RoboDK station: bokssim.rdk

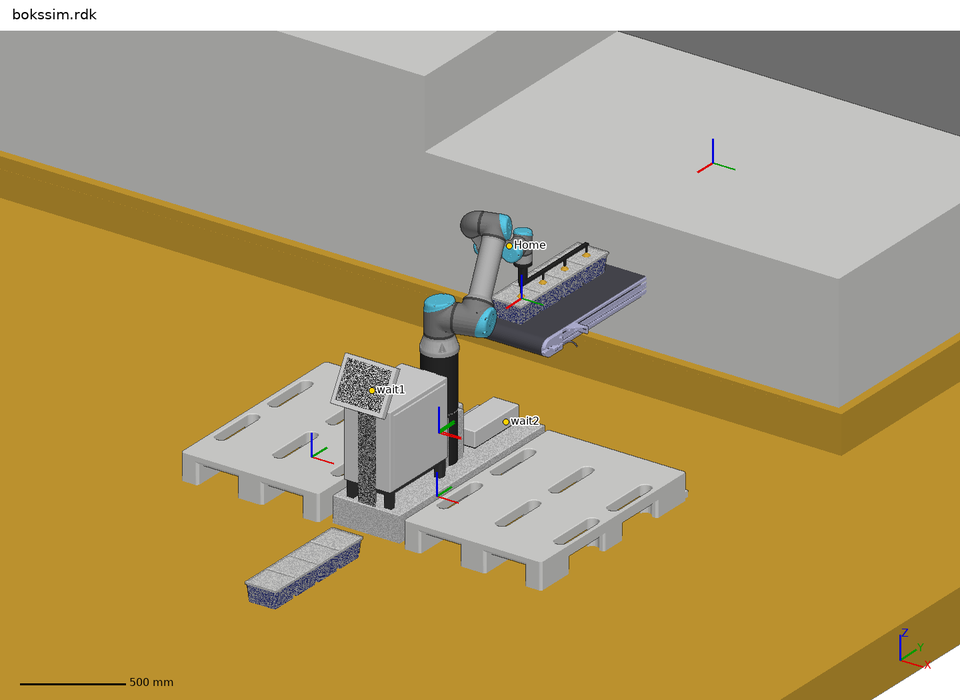
[picture v0: the station drawn from its stored meshes, robots at their saved joint values, targets as dots, program paths as lines]
Station robotsim1. Poses are relative to the parent item; angles as X-Y-Z fixed-axis rotations.
  - object pallPlast-v2 at (-1010, 360, 0) mm, size 800 x 1200 x 150 mm, geometry from pallPlast-v2.step
  - frame Conveyor Belt Base at (-200, 3610, 605) mm, rotated rx 0 ry 0 rz -90 deg
    - robot Conveyor Belt: 1 axes
        modified DH rows (alpha deg, a mm, theta deg, d mm): 0, 0, 0, 0 linear
        base shift (0, 0, 0) mm, rotated rx 0 ry 90 rz 0 deg
        joint limits [-500000] to [500000]; home [0]; saved at [0]
  - object pallPlast-v2 at (280, 360, 0) mm, size 800 x 1200 x 150 mm, geometry from pallPlast-v2.step
  - frame UR16e Base at (40, 1000, 300) mm
    - frame placeFrame at (-380, -510, -40) mm
    - frame placeFrame2 at (350, -520, -40) mm
    - object main041119-v2-v2 at (-195, 595, -300) mm, size 2050.3 x 1281 x 896.7 mm, geometry from main041119-v2-v2.step
    - target Home (Cartesian target) at (57.66, 497.76, 792.55) mm, rotated rx -180 ry 0 rz 13.73 deg; joints [103.73, -90, -90, -90, 90, 0] of UR16e
    - frame pickFrame at (-20, 711.26, 408.43) mm, rotated rx 0 ry 0 rz -90 deg
      - object fireien at (-80, 61.26, -91.57) mm, rotated rx 0 ry 0 rz -90 deg, size 180 x 720 x 110.5 mm, geometry from fireien.step
    - target wait2 (Cartesian target) at (356.79, 41.69, 130) mm, rotated rx -179.94 ry 0.02 rz -92.93 deg; joints [34.58, -172.159, -146.131, 48.35, 89.98, 37.51] of UR16e
    - target wait1 (Cartesian target) at (-356.2, -45.46, 130) mm, rotated rx -179.95 ry 0.01 rz 87.68 deg; joints [215.197, -172.165, -146.141, 48.353, 89.981, 37.517] of UR16e
  - frame Heis Base at (40, 1000, 290) mm
    - target Target 3 (Cartesian target) at (0, 0, 640) mm; joints [440] of Heis
    - target Target 4 (Cartesian target) at (0, 0, 780) mm; joints [620] of Heis
    - target Target 5 (Cartesian target) at (0, 0, 960) mm; joints [800] of Heis
    - robot Heis: 1 axes
        modified DH rows (alpha deg, a mm, theta deg, d mm): 0, 0, 0, 0 linear
        base shift (0, 0, 0) mm, rotated rx 0 ry 0 rz 90 deg
        joint limits [0] to [900]; home [0]; saved at [440]
      - tool stolpe-v2, TCP at (0, 0, 200) mm, size 180 x 180 x 700 mm, geometry from stolpe-v2.step
      - robot UR16e: 6 axes, payload 16 kg, reach 900 mm, repeatability 0.05 mm, weight 33.1 kg
          modified DH rows (alpha deg, a mm, theta deg, d mm): 0, 0, 0, 180.7; 90, 0, 180, 0; 0, 478.4, 0, 0; 0, 360, 0, 174.15; -90, 0, 0, 119.85; 90, 0, 180, 116.55
          joint limits [-360, -360, -360, -360, -360, -360] to [360, 360, 360, 360, 360, 360]; home [0, -90, -90, 0, 90, 0]; saved at [105.555, -132.207, -91.793, -46, 90, 15.555]
        - tool verkt, TCP at (0, 10, 190) mm, size 591.3 x 90 x 190.7 mm, geometry from verktøyLitenBoxFirev2.step
  - object AVD_Sjokko_SjokkPall2018_Utsnitt at (-66000, -40000, 0) mm, size 13177.1 x 13563.5 x 2830.1 mm, geometry from AVD_Sjokko_SjokkPall2018_Utsnitt.iges
  - object fireien at (0, 0, 0) mm, size 180 x 720 x 110.5 mm, geometry from fireien.step
